// EXAMPLE: Customised FB_IODEV_BASE for 2 DI, 4 AI, 2 DO and 2 AO.
//          Overloaded M_UserConfigure() method for User Configuration of channels.
FUNCTION_BLOCK FB_SENS_2_4A_2R_USER_CONFIG EXTENDS FB_IODEV_BASE
VAR_INPUT
END_VAR
VAR_OUTPUT
END_VAR
VAR
	// Control parameters as in T_IODEV_CTRL
	{attribute 'OPC.UA.DA' := '1'}
	ctrl:	T_IODEV_CTRL;	
	// Status parameters that EXTEND T_IODEV_STAT
	{attribute 'OPC.UA.DA' := '1'}
	{attribute 'OPC.UA.DA.Access' := '1'}
	stat:	T_IODEV_STAT_2_4A_2R;	
END_VAR

//
// TODO_USER
//
//
// Set References
RefCtrl	REF=ctrl;
RefStat	REF=stat;

// Set number of channels for each type.
// Default values are set to zero.
// Set whatever is not zero, i.e. whatever is defined.
// WARNING: The values MUST match the sizes of corresponding arrays above !!!
//
cfg.nNum_DI		:=	2; 	// Number of digital INPUT signals,      arrDI:	ARRAY [0..1]
cfg.nNum_AI		:=	4; 	// Number of analog INT  INPUT signals,  arrAI:	ARRAY [0..3]
cfg.nNum_RI		:=	2; 	// Number of analog REAL INPUT signals,  arrRI:	ARRAY [0..3]


//
// Set pointers for EXISTING arrays ONLY, e.g. arrDI, arrAI, etc.
//
pArrDI	:= ADR(stat.arrDI[0]);
pArrAI	:= ADR(stat.arrAI[0]);
pArrRI	:= ADR(stat.arrRI[0]);

//
// Execute the base class object FB_IODEV_BASE
//
SUPER^();

// TODO_USER
//
// Define individual channel configurations, if used.
METHOD M_UserConfigure
VAR_INPUT
END_VAR
// TODO_USER
//
// Example implementation.
// Hard code any signal configuration.
//

// Configuration parameter cfg.bUserConfig defines if 
// the hard-coded configuration below should be used or
// the signals will be configured from the WS.

//
// Digital signals
//
// Digital inputs (defined in stat structure T_IODEV_STAT_CUSTOM)
// Signal DI[0] is a door open signal
// Signal DI[1] is a light switch signal
stat.arrDI[0].M_Configure('CLOSED', 'OPEN');
stat.arrDI[1].M_Configure('OFF',    'ON');


//
// Analog signals
//
// Analog inputs of type INT (defined in stat structure T_IODEV_STAT_2_4A_2R)
stat.arrAI[0].M_Configure(CONVERSION_IODEV_NONE, 		0.0,   0.0, 0.0);
stat.arrAI[1].M_Configure(CONVERSION_IODEV_LINEAR, 		2.0,   1.0, 0.0);
stat.arrAI[2].M_Configure(CONVERSION_IODEV_QUADRATIC,	2.0,   1.0, 5.0);
// Edwards pressure guage
// P =10^(1.5*V - 12)    [mbar]
// 16-bit A/D converter, +=10V, e.g. EL3102.
// 1V = 2^16/10/2 = 3276.8 bit
// P = 10^(1.5*V - 12) = 10^(1.5/3276.8*bit - 12) = 10^(0.000457763*bit - 12)
stat.arrAI[3].M_Configure(CONVERSION_IODEV_EXP10, 	0.000457763, -12.0, 0.0);	



//
// Analog inputs of type REAL (defined in stat structure T_IODEV_STAT_2_4A_2R)
//
stat.arrRI[0].M_Configure(CONVERSION_IODEV_NONE, 		0.0,   0.0, 0.0);
stat.arrRI[1].M_Configure(CONVERSION_IODEV_LINEAR, 		2.0,   1.0, 0.0);
END_METHOD

END_FUNCTION_BLOCK

(* stored: Version 1.1.0.1, ProductVersion 3.1.4022.16
   POU FB_SENS_2_4A_2R_USER_CONFIG: Id {dfe50027-58ef-4985-85c2-ff4af7d8a8ec}, SpecialFunc None
   Method M_UserConfigure: Id {2ed1252c-6321-4945-8861-2399aae3566a} *)
